TYPE ST_ITC_RDR :
(**************************************************************************************
* 	Application		:	BoxControl Framework
*	Revision		:	$Revision: 404529 $
*	Revision date	:	$Date: 2018-04-23 08:21:38 +0200 (Mo., 23 Apr 2018) $
*	Last changed by	:	$Author: b7bolm $
*	URL				:	$URL: http://almscdc.swisslog.com/repo/SWPD/Development/BoxControlFramework/20_Release/trunk/01_Software/BCF/BCF/JumpStart/20_Product/10_App/11_Com/10_Lib/10_Conv/11_ITC/01_DUTs/ST_ITC_RDR.TcDUT $
*
*	Purpose			:	RDR Structure
*
* ------------------------------------------------------------------------------------
*	Copyright Swisslog [IP AG], Switzerland. All rights reserved.
* 
* ------------------------------------------------------------------------------------
*	
* 	Revision History: 
*
* 	VERSION			DATE			INITIALS			DESCRIPTION
*	0.1				04.01.2016		Kay Röder			Initial programming
*
**************************************************************************************)

STRUCT
	Position				: STRING(Conveyor.POSITION_STRINGLENGTH); // 12 Digit SIS Location MM-GGG-EEEE-LLL 
	CommandDataIndex		: DINT;
	AssignmentID			: UDINT;
	GroupID					: ULINT;
	ReturnCode				: E_ErrorConv;
END_STRUCT
END_TYPE

(* stored: Version 1.1.0.1, ProductVersion 3.1.4022.12
   DUT ST_ITC_RDR: Id {c90d78d1-6435-461c-a052-b36090d41849} *)
